ABB RAPID module: MAINMODULE.mod

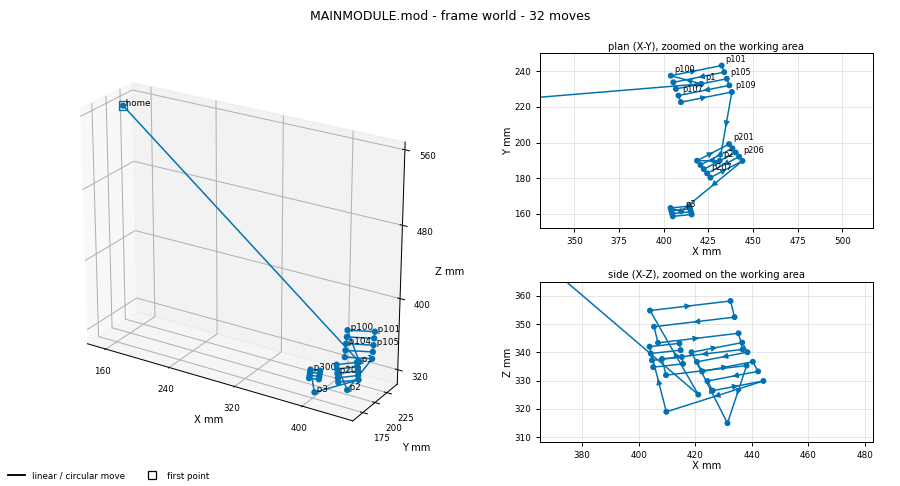
[picture p0: tool path of MAINMODULE.mod in frame world, 32 of 32 moves have a stored position in this frame; points joined in program order, loops and branches not executed]
    MODULE MainModule
    VAR robtarget home:= [[150.1, 210.4, 556.8],[0.0, 0.35559,-0.93464, 0.0],[-1,-1,0,0],[9E+09,9E+09,9E+09,9E+09,9E+09,9E+09]];
    VAR robtarget p0:= [[400, 180, 400], [0.0, 0.35559,-0.93464, 0.0], [-1,-1,0,0],[9E+09,9E+09,9E+09,9E+09,9E+09,9E+09]];
    VAR robtarget p1:= [[421.07531414201355, 232.84557667482744, 325.03671532424937], [0.0, 0.35559,-0.93464, 0.0], [-1,-1,0,0],[9E+09,9E+09,9E+09,9E+09,9E+09,9E+09]];
    VAR robtarget p100:= [[403.98480597582756, 237.40941488135263, 354.76754927845235], [0.0, 0.35559,-0.93464, 0.0], [-1,-1,0,0],[9E+09,9E+09,9E+09,9E+09,9E+09,9E+09]];
    VAR robtarget p101:= [[432.4856562678552, 243.10559166280112, 358.15690598657886], [0.0, 0.35559,-0.93464, 0.0], [-1,-1,0,0],[9E+09,9E+09,9E+09,9E+09,9E+09,9E+09]];
    VAR robtarget p102:= [[433.90569777794127, 239.3996283641764, 352.4441498324458], [0.0, 0.35559,-0.93464, 0.0], [-1,-1,0,0],[9E+09,9E+09,9E+09,9E+09,9E+09,9E+09]];
    VAR robtarget p103:= [[405.40484748591365, 233.70345158272792, 349.05479312431925], [0.0, 0.35559,-0.93464, 0.0], [-1,-1,0,0],[9E+09,9E+09,9E+09,9E+09,9E+09,9E+09]];
    VAR robtarget p104:= [[406.82488899599974, 229.9974882841032, 343.3420369701861], [0.0, 0.35559,-0.93464, 0.0], [-1,-1,0,0],[9E+09,9E+09,9E+09,9E+09,9E+09,9E+09]];
    VAR robtarget p105:= [[435.32573928802736, 235.69366506555167, 346.73139367831266], [0.0, 0.35559,-0.93464, 0.0], [-1,-1,0,0],[9E+09,9E+09,9E+09,9E+09,9E+09,9E+09]];
    VAR robtarget p106:= [[436.74578079811346, 231.98770176692696, 341.01863752417955], [0.0, 0.35559,-0.93464, 0.0], [-1,-1,0,0],[9E+09,9E+09,9E+09,9E+09,9E+09,9E+09]];
    VAR robtarget p107:= [[408.24493050608584, 226.29152498547847, 337.629280816053], [0.0, 0.35559,-0.93464, 0.0], [-1,-1,0,0],[9E+09,9E+09,9E+09,9E+09,9E+09,9E+09]];
    VAR robtarget p108:= [[409.66497201617193, 222.58556168685377, 331.9165246619199], [0.0, 0.35559,-0.93464, 0.0], [-1,-1,0,0],[9E+09,9E+09,9E+09,9E+09,9E+09,9E+09]];
    VAR robtarget p109:= [[438.16582230819955, 228.28173846830225, 335.3058813700464], [0.0, 0.35559,-0.93464, 0.0], [-1,-1,0,0],[9E+09,9E+09,9E+09,9E+09,9E+09,9E+09]];
    VAR robtarget p2:= [[431.3907785964209, 189.75018373039583, 314.9354023856076], [0.0, 0.35559,-0.93464, 0.0], [-1,-1,0,0],[9E+09,9E+09,9E+09,9E+09,9E+09,9E+09]];
    VAR robtarget p200:= [[418.6786763166023, 189.79896272027838, 340.0113735016163], [0.0, 0.35559,-0.93464, 0.0], [-1,-1,0,0],[9E+09,9E+09,9E+09,9E+09,9E+09,9E+09]];
    VAR robtarget p201:= [[436.60094993086255, 199.13063315087797, 343.4340310907879], [0.0, 0.35559,-0.93464, 0.0], [-1,-1,0,0],[9E+09,9E+09,9E+09,9E+09,9E+09,9E+09]];
    VAR robtarget p202:= [[438.4764326672068, 196.77332604828678, 340.04038113549063], [0.0, 0.35559,-0.93464, 0.0], [-1,-1,0,0],[9E+09,9E+09,9E+09,9E+09,9E+09,9E+09]];
    VAR robtarget p203:= [[420.5541590529466, 187.44165561768722, 336.617723546319], [0.0, 0.35559,-0.93464, 0.0], [-1,-1,0,0],[9E+09,9E+09,9E+09,9E+09,9E+09,9E+09]];
    VAR robtarget p204:= [[422.42964178929077, 185.08434851509605, 333.22407359102175], [0.0, 0.35559,-0.93464, 0.0], [-1,-1,0,0],[9E+09,9E+09,9E+09,9E+09,9E+09,9E+09]];
    VAR robtarget p205:= [[440.351915403551, 194.41601894569564, 336.64673118019346], [0.0, 0.35559,-0.93464, 0.0], [-1,-1,0,0],[9E+09,9E+09,9E+09,9E+09,9E+09,9E+09]];
    VAR robtarget p206:= [[442.2273981398952, 192.05871184310448, 333.25308122489616], [0.0, 0.35559,-0.93464, 0.0], [-1,-1,0,0],[9E+09,9E+09,9E+09,9E+09,9E+09,9E+09]];
    VAR robtarget p207:= [[424.305124525635, 182.7270414125049, 329.8304236357245], [0.0, 0.35559,-0.93464, 0.0], [-1,-1,0,0],[9E+09,9E+09,9E+09,9E+09,9E+09,9E+09]];
    VAR robtarget p208:= [[426.1806072619792, 180.3697343099137, 326.4367736804272], [0.0, 0.35559,-0.93464, 0.0], [-1,-1,0,0],[9E+09,9E+09,9E+09,9E+09,9E+09,9E+09]];
    VAR robtarget p209:= [[444.10288087623945, 189.7014047405133, 329.8594312695989], [0.0, 0.35559,-0.93464, 0.0], [-1,-1,0,0],[9E+09,9E+09,9E+09,9E+09,9E+09,9E+09]];
    VAR robtarget p3:= [[409.75944685253, 161.52375315307398, 318.95746954718817], [0.0, 0.35559,-0.93464, 0.0], [-1,-1,0,0],[9E+09,9E+09,9E+09,9E+09,9E+09,9E+09]];
    VAR robtarget p300:= [[403.8436760397758, 163.35144322201327, 341.9930354525497], [0.0, 0.35559,-0.93464, 0.0], [-1,-1,0,0],[9E+09,9E+09,9E+09,9E+09,9E+09,9E+09]];
    VAR robtarget p301:= [[414.4023421763141, 164.39235910663356, 343.17245217568313], [0.0, 0.35559,-0.93464, 0.0], [-1,-1,0,0],[9E+09,9E+09,9E+09,9E+09,9E+09,9E+09]];
    VAR robtarget p302:= [[414.8266340059708, 162.82692709913394, 340.7556026643976], [0.0, 0.35559,-0.93464, 0.0], [-1,-1,0,0],[9E+09,9E+09,9E+09,9E+09,9E+09,9E+09]];
    VAR robtarget p303:= [[404.26796786943254, 161.78601121451368, 339.5761859412642], [0.0, 0.35559,-0.93464, 0.0], [-1,-1,0,0],[9E+09,9E+09,9E+09,9E+09,9E+09,9E+09]];
    VAR robtarget p304:= [[404.6922596990892, 160.22057920701405, 337.15933642997874], [0.0, 0.35559,-0.93464, 0.0], [-1,-1,0,0],[9E+09,9E+09,9E+09,9E+09,9E+09,9E+09]];
    VAR robtarget p305:= [[415.2509258356275, 161.26149509163432, 338.3387531531122], [0.0, 0.35559,-0.93464, 0.0], [-1,-1,0,0],[9E+09,9E+09,9E+09,9E+09,9E+09,9E+09]];
    VAR robtarget p306:= [[415.67521766528426, 159.6960630841347, 335.92190364182665], [0.0, 0.35559,-0.93464, 0.0], [-1,-1,0,0],[9E+09,9E+09,9E+09,9E+09,9E+09,9E+09]];
    VAR robtarget p307:= [[405.1165515287459, 158.65514719951443, 334.7424869186932], [0.0, 0.35559,-0.93464, 0.0], [-1,-1,0,0],[9E+09,9E+09,9E+09,9E+09,9E+09,9E+09]];
    PERS tooldata tool1:=  [TRUE, [ [0, 0, 100], [1, 0, 0 ,0] ], [0.001, [0, 0, 0.001], [1, 0, 0, 0], 0, 0, 0]];
    PERS wobjdata DefaultWObj;

    PROC main()
        MoveL home, v50, z50, tool1;
        MoveL p1, v50, z50, tool1;
        WaitTime 3;
        MoveL p100, v50, z50, tool1;
        MoveL p101, v50, z50, tool1;
        MoveL p102, v50, z50, tool1;
        MoveL p103, v50, z50, tool1;
        MoveL p104, v50, z50, tool1;
        MoveL p105, v50, z50, tool1;
        MoveL p106, v50, z50, tool1;
        MoveL p107, v50, z50, tool1;
        MoveL p108, v50, z50, tool1;
        MoveL p109, v50, z50, tool1;
        WaitTime 3;
        MoveL p2, v50, z50, tool1;
        WaitTime 3;
        MoveL p200, v50, z50, tool1;
        MoveL p201, v50, z50, tool1;
        MoveL p202, v50, z50, tool1;
        MoveL p203, v50, z50, tool1;
        MoveL p204, v50, z50, tool1;
        MoveL p205, v50, z50, tool1;
        MoveL p206, v50, z50, tool1;
        MoveL p207, v50, z50, tool1;
        MoveL p208, v50, z50, tool1;
        MoveL p209, v50, z50, tool1;
        WaitTime 3;
        MoveL p3, v50, z50, tool1;
        WaitTime 3;
        MoveL p300, v50, z50, tool1;
        MoveL p301, v50, z50, tool1;
        MoveL p302, v50, z50, tool1;
        MoveL p303, v50, z50, tool1;
        MoveL p304, v50, z50, tool1;
        MoveL p305, v50, z50, tool1;
        MoveL p306, v50, z50, tool1;
        MoveL p307, v50, z50, tool1;
        WaitTime 3;
    ENDPROC
ENDMODULE
